PROGRAM MAIN
VAR
	ConfigRoot : FB_ConfigRoot;
END_VAR

ConfigRoot.Run();

END_PROGRAM

(* stored: Version 1.1.0.1, ProductVersion 3.1.4026.18
   POU MAIN: Id {6a544a39-0af3-40f7-b9b9-87a109cea42a}, SpecialFunc None *)
